// TIA Portal V21 export
// export: Created 2026-06-08T02:43:13.3990248Z, ExportSetting WithReadOnly, DisplayName Totally Integrated Automation Portal, DisplayVersion V21, DisplayName SINAMICS Startdrive Advanced, DisplayVersion V21, DisplayName SINAMICS Startdrive G110M, G120, G120C, G120D, G120P, G115D, DisplayVersion V21, DisplayName SINAMICS Startdrive G130, G150, S120, S150, G200, G220, S200, S210, S220, Innomotics MVD, DisplayVersion V21, DisplayName STEP 7 Professional, DisplayVersion V21, DisplayName STEP 7 Safety, DisplayVersion V21, DisplayName Tech WebApplication, DisplayVersion V21, DisplayName WinCC Basic/Comfort/Advanced, DisplayVersion V21, DisplayName WinCC Professional, DisplayVersion V21, DisplayName WinCC Unified, DisplayVersion V21
ORGANIZATION_BLOCK "Main"   // OB1, LAD, ProgramCycle
TITLE = "Main Program Sweep (Cycle)"
{ S7_Optimized_Access := 'TRUE' }
// stored: CodeModifiedDate 2026-06-07T02:45:42.286589Z, CompileDate 2026-06-07T02:45:42.286589Z, ConstantName OB_Main, CreationDate 2026-05-21T06:56:38.8521971Z, DownloadDate 2026-06-07T02:47:24.9117008Z, EventClass Program cycle, InterfaceModifiedDate 2008-07-21T16:55:08.419547Z, IsConsistent true, LoadMemoryLength 4577, ModifiedDate 2026-06-07T02:45:42.286589Z, PLCSimAdvancedSupport true, ParameterModified 2008-07-21T16:55:08.419547Z, PriorityNumber 1, ProcessImagePartNumber 65535, SetENOAutomatically false, StructureModified 2008-07-21T16:55:08.419547Z, WorkMemoryLength 40
   VAR_INPUT
      Initial_Call : Bool;
      Remanence : Bool;
   END_VAR
   VAR_TEMP
      Temp_Target_F : Real;
      Temp_Target_A : Real;
      hbRead : Int;   // 心跳快照（防异步刷新）
   END_VAR
BEGIN

REGION Network 1 (SCL): 心跳快照（防异步刷新）
   // SCL 转换逻辑
   "FC_CallFertigationControl"();
END_REGION
END_ORGANIZATION_BLOCK
